DATA_BLOCK "IDB_LineC1"   // DB10
// stored: InstanceOfName LineC1.FB_LineC1, InstanceOfType FB, Namespace LineC1
"LineC1.FB_LineC1"
   // VAR
   //    "Conveyor_C1.1.1" : "Global.FB_Conveyor";
   //    "Conveyor_C1.1.2" { S7_SetPoint := 'True'} : "Global.FB_Conveyor";
   //    "Conveyor_C1.1.3" { S7_SetPoint := 'True'} : "Global.FB_Conveyor";
   //    "MABS_C1.2.1" : "Global.FB_MABS";
   //    "MABS_C1.2.2" { S7_SetPoint := 'True'} : "Global.FB_MABS";
   //    "Conveyor_C1.3.1" { S7_SetPoint := 'True'} : "Global.FB_Conveyor";
   //    "Conveyor_C1.3.2" { S7_SetPoint := 'True'} : "Global.FB_Conveyor";
   //    "Conveyor_C1.3.3" { S7_SetPoint := 'True'} : "Global.FB_Conveyor";
   //    "Conveyor_C1.3.4" { S7_SetPoint := 'True'} : "Global.FB_Conveyor";
   //    "Conveyor_C1.3.5" { S7_SetPoint := 'True'} : "Global.FB_Conveyor";
   //    "Conveyor_C1.3.6" { S7_SetPoint := 'True'} : "Global.FB_Conveyor";
   //    "Conveyor_C1.3.7" { S7_SetPoint := 'True'} : "Global.FB_Conveyor";
   //    "Conveyor_C1.3.8" { S7_SetPoint := 'True'} : "Global.FB_Conveyor";
   //    "Conveyor_C1.3.9" { S7_SetPoint := 'True'} : "Global.FB_Conveyor";
   //    "Conveyor_C1.3.10" { S7_SetPoint := 'True'} : "Global.FB_Conveyor";
   //    "Conveyor_C1.4.1" { S7_SetPoint := 'True'} : "Global.FB_Conveyor";
   //    "Conveyor_C1.4.2" { S7_SetPoint := 'True'} : "Global.FB_Conveyor";
   //    "Conveyor_C1.4.3" { S7_SetPoint := 'True'} : "Global.FB_Conveyor";
   //    "Conveyor_C1.4.4" { S7_SetPoint := 'True'} : "Global.FB_Conveyor";
   //    "Conveyor_C1.5.1" { S7_SetPoint := 'True'} : "Global.FB_Conveyor";
   //    "Conveyor_C1.6.1" { S7_SetPoint := 'True'} : "Global.FB_Conveyor";
   //    "Conveyor_C1.6.2" { S7_SetPoint := 'True'} : "Global.FB_Conveyor";
   //    "Conveyor_C1.7.1" { S7_SetPoint := 'True'} : "Global.FB_Conveyor";
   //    "Conveyor_C1.7.2" { S7_SetPoint := 'True'} : "Global.FB_Conveyor";
   //    "Conveyor_C1.7.3" { S7_SetPoint := 'True'} : "Global.FB_Conveyor";
   //    "Conveyor_C1.7.4" { S7_SetPoint := 'True'} : "Global.FB_Conveyor";
   //    "Conveyor_C1.7.5" { S7_SetPoint := 'True'} : "Global.FB_Conveyor";
   //    "Conveyor_C1.7.6" { S7_SetPoint := 'True'} : "Global.FB_Conveyor";
   //    "Conveyor_C1.7.7" { S7_SetPoint := 'True'} : "Global.FB_Conveyor";
   //    "Conveyor_C1.7.8" { S7_SetPoint := 'True'} : "Global.FB_Conveyor";
   //    "Conveyor_C1.7.9" { S7_SetPoint := 'True'} : "Global.FB_Conveyor";
   //    "Conveyor_C1.7.10" { S7_SetPoint := 'True'} : "Global.FB_Conveyor";
   //    "Conveyor_C1.8.0" { S7_SetPoint := 'True'} : "Global.FB_Conveyor";
   //    "Conveyor_C1.9.1" { S7_SetPoint := 'True'} : "Global.FB_Conveyor";
   //    "Conveyor_C1.10.1" { S7_SetPoint := 'True'} : "Global.FB_Conveyor";
   //    "Conveyor_C1.11.1" { S7_SetPoint := 'True'} : "Global.FB_Conveyor";
   //    "Conveyor_C1.11.2" { S7_SetPoint := 'True'} : "Global.FB_Conveyor";
   //    "Conveyor_C1.12.1" { S7_SetPoint := 'True'} : "Global.FB_Conveyor";
   //    "Conveyor_C1.12.2" { S7_SetPoint := 'True'} : "Global.FB_Conveyor";
   //    "Conveyor_C1.12.3" { S7_SetPoint := 'True'} : "Global.FB_Conveyor";
   //    "Transfer_C1.13.1" : "Global.FB_S300_tTransMode";
   //    "Transfer_C1.14.1" { S7_SetPoint := 'True'} : "Global.FB_S300_tTransMode";
   //    "Conveyor_C1.15.2" { S7_SetPoint := 'True'} : "Global.FB_Conveyor";
   //    "Conveyor_C1.15.3" { S7_SetPoint := 'True'} : "Global.FB_Conveyor";
   //    "Conveyor_C1.15.4" { S7_SetPoint := 'True'} : "Global.FB_Conveyor";
   //    "Conveyor_C1.16.1" { S7_SetPoint := 'True'} : "Global.FB_Conveyor";
   //    "Conveyor_C1.17.0" { S7_SetPoint := 'True'} : "Global.FB_Conveyor";
   //    "Conveyor_C1.18.1" { S7_SetPoint := 'True'} : "Global.FB_Conveyor";
   //    "Conveyor_C1.18.2" { S7_SetPoint := 'True'} : "Global.FB_Conveyor";
   //    "Conveyor_C1.18.3" { S7_SetPoint := 'True'} : "Global.FB_Conveyor";
   //    "Conveyor_C1.18.4" { S7_SetPoint := 'True'} : "Global.FB_Conveyor";
   //    "Conveyor_C1.18.5" { S7_SetPoint := 'True'} : "Global.FB_Conveyor";
   //    "Conveyor_C1.18.6" { S7_SetPoint := 'True'} : "Global.FB_Conveyor";
   //    "Conveyor_C1.18.7" { S7_SetPoint := 'True'} : "Global.FB_Conveyor";
   //    "Conveyor_C1.19.1" { S7_SetPoint := 'True'} : "Global.FB_Conveyor";
   //    "Conveyor_C1.20.2" { S7_SetPoint := 'True'} : "Global.FB_Conveyor";
   // END_VAR
BEGIN
END_DATA_BLOCK

DATA_BLOCK "IDB_LineD1"   // DB11
// stored: InstanceOfName LineD1.FB_LineD1, InstanceOfType FB, Namespace LineD1
"LineD1.FB_LineD1"
   // VAR
   //    "Conveyor_D1.1.1" : "Global.FB_Conveyor";
   //    "MABS_D1.1.1" : "Global.FB_MABS";
   //    "Transfer_D1.1.1" : "Global.FB_S300_tTransMode";
   // END_VAR
BEGIN
END_DATA_BLOCK

DATA_BLOCK "IDB_EmptyLine"   // DB9
// stored: InstanceOfName EmptyLine.FB_EmptyLine, InstanceOfType FB, Namespace EmptyLine
"EmptyLine.FB_EmptyLine"
   // VAR
   //    "J1.1.1" : "Global.FB_Conveyor";
   //    "J1.1.2" { S7_SetPoint := 'True'} : "Global.FB_Conveyor";
   //    "J1.1.3" { S7_SetPoint := 'True'} : "Global.FB_Conveyor";
   //    "J1.1.4" { S7_SetPoint := 'True'} : "Global.FB_Conveyor";
   //    "J1.1.5" { S7_SetPoint := 'True'} : "Global.FB_Conveyor";
   //    "J1.1.6" { S7_SetPoint := 'True'} : "Global.FB_Conveyor";
   //    "J1.1.7" { S7_SetPoint := 'True'} : "Global.FB_Conveyor";
   //    "J1.1.8" { S7_SetPoint := 'True'} : "Global.FB_Conveyor";
   //    "J1.1.9" { S7_SetPoint := 'True'} : "Global.FB_Conveyor";
   //    "J1.1.10" { S7_SetPoint := 'True'} : "Global.FB_Conveyor";
   //    "J1.1.11" { S7_SetPoint := 'True'} : "Global.FB_Conveyor";
   //    "J1.1.12" { S7_SetPoint := 'True'} : "Global.FB_Conveyor";
   //    "J1.1.13" { S7_SetPoint := 'True'} : "Global.FB_Conveyor";
   //    "J1.1.14" { S7_SetPoint := 'True'} : "Global.FB_Conveyor";
   //    "J1.1.15" { S7_SetPoint := 'True'} : "Global.FB_Conveyor";
   //    "J1.1.16" { S7_SetPoint := 'True'} : "Global.FB_Conveyor";
   //    "J1.2.1" { S7_SetPoint := 'True'} : "Global.FB_Conveyor";
   //    "J1.2.2" { S7_SetPoint := 'True'} : "Global.FB_Conveyor";
   //    "J1.2.3" { S7_SetPoint := 'True'} : "Global.FB_Conveyor";
   //    "J2.1.1" { S7_SetPoint := 'True'} : "Global.FB_Conveyor";
   //    "J2.1.2" { S7_SetPoint := 'True'} : "Global.FB_Conveyor";
   //    "J2.1.3" { S7_SetPoint := 'True'} : "Global.FB_Conveyor";
   //    "J2.1.4" { S7_SetPoint := 'True'} : "Global.FB_Conveyor";
   //    "J2.1.5" { S7_SetPoint := 'True'} : "Global.FB_Conveyor";
   //    "J2.1.6" { S7_SetPoint := 'True'} : "Global.FB_Conveyor";
   //    "J2.1.7" { S7_SetPoint := 'True'} : "Global.FB_Conveyor";
   //    "J2.1.8" { S7_SetPoint := 'True'} : "Global.FB_Conveyor";
   //    "J2.1.9" { S7_SetPoint := 'True'} : "Global.FB_Conveyor";
   //    "J2.1.10" { S7_SetPoint := 'True'} : "Global.FB_Conveyor";
   //    "J2.1.11" { S7_SetPoint := 'True'} : "Global.FB_Conveyor";
   //    "J2.1.12" { S7_SetPoint := 'True'} : "Global.FB_Conveyor";
   //    "J2.1.13" { S7_SetPoint := 'True'} : "Global.FB_Conveyor";
   //    "J2.1.14" { S7_SetPoint := 'True'} : "Global.FB_Conveyor";
   //    "J2.1.15" { S7_SetPoint := 'True'} : "Global.FB_Conveyor";
   //    "J2.2.1" { S7_SetPoint := 'True'} : "Global.FB_Conveyor";
   //    "J2.2.2" { S7_SetPoint := 'True'} : "Global.FB_Conveyor";
   //    "J2.3.1" { S7_SetPoint := 'True'} : "Global.FB_Conveyor";
   //    "J2.4.1" { S7_SetPoint := 'True'} : "Global.FB_Conveyor";
   //    "J1.2.4" { S7_SetPoint := 'True'} : "Global.FB_Conveyor";
   //    "J1.2.5" { S7_SetPoint := 'True'} : "Global.FB_Conveyor";
   //    "J1.3.1" { S7_SetPoint := 'True'} : "Global.FB_Conveyor";
   //    "J1.3.2" { S7_SetPoint := 'True'} : "Global.FB_Conveyor";
   //    "J1.4.1" { S7_SetPoint := 'True'} : "Global.FB_Conveyor";
   //    "J1.4.2" { S7_SetPoint := 'True'} : "Global.FB_Conveyor";
   //    "J1.4.3" { S7_SetPoint := 'True'} : "Global.FB_Conveyor";
   //    "J1.4.4" { S7_SetPoint := 'True'} : "Global.FB_Conveyor";
   //    "J1.4.5" { S7_SetPoint := 'True'} : "Global.FB_Conveyor";
   //    "J1.4.6" { S7_SetPoint := 'True'} : "Global.FB_Conveyor";
   //    "J1.4.7" { S7_SetPoint := 'True'} : "Global.FB_Conveyor";
   //    "J1.5.1" { S7_SetPoint := 'True'} : "Global.FB_Conveyor";
   //    "J1.5.2" { S7_SetPoint := 'True'} : "Global.FB_Conveyor";
   //    "J1.5.3" { S7_SetPoint := 'True'} : "Global.FB_Conveyor";
   //    "J1.5.4" { S7_SetPoint := 'True'} : "Global.FB_Conveyor";
   //    "J1.6.1" { S7_SetPoint := 'True'} : "Global.FB_MABS";
   //    "J1.6.2" { S7_SetPoint := 'True'} : "Global.FB_MABS";
   //    "J1.7.1" { S7_SetPoint := 'True'} : "Global.FB_Conveyor";
   //    "J1.7.2" { S7_SetPoint := 'True'} : "Global.FB_Conveyor";
   //    "J1.8.1" { S7_SetPoint := 'True'} : "Global.FB_Conveyor";
   //    "J1.8.2" { S7_SetPoint := 'True'} : "Global.FB_Conveyor";
   //    "J1.9.1" { S7_SetPoint := 'True'} : "Global.FB_Conveyor";
   //    "J1.10.1" { S7_SetPoint := 'True'} : "Global.FB_Conveyor";
   //    "J1.11.1" { S7_SetPoint := 'True'} : "Global.FB_Conveyor";
   //    "J1.11.2" { S7_SetPoint := 'True'} : "Global.FB_Conveyor";
   //    "J1.11.3" { S7_SetPoint := 'True'} : "Global.FB_Conveyor";
   //    "J1.11.4" { S7_SetPoint := 'True'} : "Global.FB_Conveyor";
   //    "J1.11.5" { S7_SetPoint := 'True'} : "Global.FB_Conveyor";
   //    "J1.11.6" { S7_SetPoint := 'True'} : "Global.FB_Conveyor";
   //    "J1.11.7" { S7_SetPoint := 'True'} : "Global.FB_Conveyor";
   //    "J1.11.8" { S7_SetPoint := 'True'} : "Global.FB_Conveyor";
   //    "J1.11.9" { S7_SetPoint := 'True'} : "Global.FB_Conveyor";
   //    "J1.11.10" { S7_SetPoint := 'True'} : "Global.FB_Conveyor";
   //    "J1.11.11" { S7_SetPoint := 'True'} : "Global.FB_Conveyor";
   //    "J1.11.12" { S7_SetPoint := 'True'} : "Global.FB_Conveyor";
   //    "J1.11.13" { S7_SetPoint := 'True'} : "Global.FB_Conveyor";
   //    "K1.1.1" { S7_SetPoint := 'True'} : "Global.FB_Conveyor";
   //    "K1.2.1" { S7_SetPoint := 'True'} : "Global.FB_Conveyor";
   //    "K1.3.1" { S7_SetPoint := 'True'} : "Global.FB_Conveyor";
   //    "K1.4.1" { S7_SetPoint := 'True'} : "Global.FB_Conveyor";
   //    "K1.4.2" { S7_SetPoint := 'True'} : "Global.FB_Conveyor";
   //    "K1.4.3" { S7_SetPoint := 'True'} : "Global.FB_Conveyor";
   //    "K1.4.4" { S7_SetPoint := 'True'} : "Global.FB_Conveyor";
   //    "K1.4.5" { S7_SetPoint := 'True'} : "Global.FB_Conveyor";
   //    "K1.4.6" { S7_SetPoint := 'True'} : "Global.FB_Conveyor";
   //    "K1.4.7" { S7_SetPoint := 'True'} : "Global.FB_Conveyor";
   //    "K1.4.8" { S7_SetPoint := 'True'} : "Global.FB_Conveyor";
   //    "K1.4.9" { S7_SetPoint := 'True'} : "Global.FB_Conveyor";
   //    "K1.4.10" { S7_SetPoint := 'True'} : "Global.FB_Conveyor";
   //    "K1.5.1" { S7_SetPoint := 'True'} : "Global.FB_Conveyor";
   //    "K1.5.2" { S7_SetPoint := 'True'} : "Global.FB_Conveyor";
   //    "K1.5.3" { S7_SetPoint := 'True'} : "Global.FB_Conveyor";
   //    "K1.5.4" { S7_SetPoint := 'True'} : "Global.FB_Conveyor";
   //    "K1.5.5" { S7_SetPoint := 'True'} : "Global.FB_Conveyor";
   //    "K1.5.6" { S7_SetPoint := 'True'} : "Global.FB_Conveyor";
   //    "K1.5.7" { S7_SetPoint := 'True'} : "Global.FB_Conveyor";
   //    "K1.5.8" { S7_SetPoint := 'True'} : "Global.FB_Conveyor";
   //    "K1.6.1" { S7_SetPoint := 'True'} : "Global.FB_Conveyor";
   //    "K1.6.2" { S7_SetPoint := 'True'} : "Global.FB_Conveyor";
   //    "K1.7.1" { S7_SetPoint := 'True'} : "Global.FB_Conveyor";
   //    "K1.7.2" { S7_SetPoint := 'True'} : "Global.FB_Conveyor";
   //    "K1.8.1" { S7_SetPoint := 'True'} : "Global.FB_Conveyor";
   //    "K1.8.2" { S7_SetPoint := 'True'} : "Global.FB_Conveyor";
   //    "K1.8.3" { S7_SetPoint := 'True'} : "Global.FB_Conveyor";
   //    "K1.9.1" { S7_SetPoint := 'True'} : "Global.FB_Conveyor";
   //    "K1.9.2" { S7_SetPoint := 'True'} : "Global.FB_Conveyor";
   //    "K1.9.3" { S7_SetPoint := 'True'} : "Global.FB_Conveyor";
   //    "K1.9.4" { S7_SetPoint := 'True'} : "Global.FB_Conveyor";
   //    "K1.9.5" { S7_SetPoint := 'True'} : "Global.FB_Conveyor";
   //    "K1.9.6" { S7_SetPoint := 'True'} : "Global.FB_Conveyor";
   //    "K1.9.7" { S7_SetPoint := 'True'} : "Global.FB_Conveyor";
   //    "K1.10.1" { S7_SetPoint := 'True'} : "Global.FB_Conveyor";
   // END_VAR
BEGIN
END_DATA_BLOCK

DATA_BLOCK "IDB_GlobalStatus"   // DB48
// stored: InstanceOfName Global.FB_GlobalStatus, InstanceOfType FB, Namespace Global
"Global.FB_GlobalStatus"
   // VAR
   //    Line : Struct
   //       ProductionLine : "Global.ConveyorStatus";
   //       EmptyLine { S7_SetPoint := 'True'} : "Global.ConveyorStatus";
   //       PackedLine { S7_SetPoint := 'True'} : "Global.ConveyorStatus";
   //    END_STRUCT;
   //    cmp : Struct
   //       ProductionTotes_Value0 : Array[_.gminProductionLine.._.gmaxProductionLine] of Bool;
   //       ProductionTotes_Value1 : Array[_.gminProductionLine.._.gmaxProductionLine] of Bool;
   //       EmptyLine_Value0 : Array[_.gminEmptyLine.._.gmaxEmptyLine] of Bool;
   //       EmptyLine_Value1 : Array[_.gminEmptyLine.._.gmaxEmptyLine] of Bool;
   //       PackedLine_Value0 : Array[_.gminPackedLine.._.gmaxPackedLine] of Bool;
   //       PackedLine_Value1 : Array[_.gminPackedLine.._.gmaxPackedLine] of Bool;
   //    END_STRUCT;
   //    ForVisu : Struct
   //       Line : Struct
   //          ProductionLine : Word;
   //          EmptyLine : Word;
   //          PackedLine : Word;
   //       END_STRUCT;
   //    END_STRUCT;
   // END_VAR
BEGIN
   cmp.ProductionTotes_Value1[1001..1192] := True;
   cmp.EmptyLine_Value1[2001..2109] := True;
   cmp.PackedLine_Value1[3001..3040] := True;
END_DATA_BLOCK

DATA_BLOCK "IDB_PackedLine"   // DB10
// stored: Access Published, InstanceOfName PackedLine.FB_PackedLine, InstanceOfType FB, Namespace PackedLine
"PackedLine.FB_PackedLine"
   // VAR
   //    "G1.1.1" { S7_SetPoint := 'True'} : "Global.FB_Conveyor";
   //    "G1.1.2" { S7_SetPoint := 'True'} : "Global.FB_Conveyor";
   //    "G1.1.3" { S7_SetPoint := 'True'} : "Global.FB_Conveyor";
   //    "G1.1.4" { S7_SetPoint := 'True'} : "Global.FB_Conveyor";
   //    "G1.1.5" { S7_SetPoint := 'True'} : "Global.FB_Conveyor";
   //    "G1.1.6" { S7_SetPoint := 'True'} : "Global.FB_Conveyor";
   //    "G1.1.7" { S7_SetPoint := 'True'} : "Global.FB_Conveyor";
   //    "G1.1.8" { S7_SetPoint := 'True'} : "Global.FB_Conveyor";
   //    "G1.1.9" { S7_SetPoint := 'True'} : "Global.FB_Conveyor";
   //    "G1.1.10" { S7_SetPoint := 'True'} : "Global.FB_Conveyor";
   //    "G1.1.11" { S7_SetPoint := 'True'} : "Global.FB_Conveyor";
   //    "G1.1.12" { S7_SetPoint := 'True'} : "Global.FB_Conveyor";
   //    "G1.1.13" { S7_SetPoint := 'True'} : "Global.FB_Conveyor";
   //    "G1.1.14" { S7_SetPoint := 'True'} : "Global.FB_Conveyor";
   //    "G1.1.15" { S7_SetPoint := 'True'} : "Global.FB_Conveyor";
   //    "G1.1.16" { S7_SetPoint := 'True'} : "Global.FB_Conveyor";
   //    "G1.1.17" { S7_SetPoint := 'True'} : "Global.FB_Conveyor";
   //    "G1.1.18" { S7_SetPoint := 'True'} : "Global.FB_Conveyor";
   //    "G1.1.19" { S7_SetPoint := 'True'} : "Global.FB_Conveyor";
   //    "G1.2.1" { S7_SetPoint := 'True'} : "Global.FB_Conveyor";
   //    "G1.2.2" { S7_SetPoint := 'True'} : "Global.FB_Conveyor";
   //    "G1.3.1" { S7_SetPoint := 'True'} : "Global.FB_Conveyor";
   //    "G1.4.1" { S7_SetPoint := 'True'} : "Global.FB_Conveyor";
   //    "G1.4.2" { S7_SetPoint := 'True'} : "Global.FB_Conveyor";
   //    "G1.4.3" { S7_SetPoint := 'True'} : "Global.FB_Conveyor";
   //    "G1.4.4" { S7_SetPoint := 'True'} : "Global.FB_Conveyor";
   //    "G1.4.5" { S7_SetPoint := 'True'} : "Global.FB_Conveyor";
   //    "G1.4.6" { S7_SetPoint := 'True'} : "Global.FB_Conveyor";
   //    "G1.5.1" { S7_SetPoint := 'True'} : "Global.FB_Conveyor";
   //    "G1.5.2" { S7_SetPoint := 'True'} : "Global.FB_Conveyor";
   //    "G1.5.3" { S7_SetPoint := 'True'} : "Global.FB_Conveyor";
   //    "G1.5.4" { S7_SetPoint := 'True'} : "Global.FB_Conveyor";
   //    "G1.5.5" { S7_SetPoint := 'True'} : "Global.FB_Conveyor";
   //    "G1.5.6" { S7_SetPoint := 'True'} : "Global.FB_Conveyor";
   //    "G1.6.1" { S7_SetPoint := 'True'} : "Global.FB_Conveyor";
   //    "G1.6.2" { S7_SetPoint := 'True'} : "Global.FB_Conveyor";
   //    "G1.7.1" { S7_SetPoint := 'True'} : "Global.FB_Conveyor";
   //    "G1.7.2" { S7_SetPoint := 'True'} : "Global.FB_Conveyor";
   //    "G1.7.3" { S7_SetPoint := 'True'} : "Global.FB_Conveyor";
   //    "G1.7.4" { S7_SetPoint := 'True'} : "Global.FB_Conveyor";
   // END_VAR
BEGIN
END_DATA_BLOCK

DATA_BLOCK "IDB_Merging"   // DB27
// stored: InstanceOfName ProductionLine.FB_Merging, InstanceOfType FB, Namespace ProductionLine
"ProductionLine.FB_Merging"
   // VAR
   //    "Merge_A1.7.3" : "Global.FB_Merging";
   //    "Merge_A1.9.3" : "Global.FB_Merging";
   //    "Merge_B1.6.1" { S7_SetPoint := 'True'} : "Global.FB_Merging";
   // END_VAR
BEGIN
END_DATA_BLOCK

DATA_BLOCK "IDB_ProductionLine"   // DB8
// stored: InstanceOfName ProductionLine.FB_ProductionLine, InstanceOfType FB, Namespace ProductionLine
"ProductionLine.FB_ProductionLine"
   // VAR
   //    "A1.1.1" { S7_SetPoint := 'True'} : "Global.FB_Conveyor";
   //    "A1.1.2" { S7_SetPoint := 'True'} : "Global.FB_Conveyor";
   //    "A1.1.3" { S7_SetPoint := 'True'} : "Global.FB_Conveyor";
   //    "A1.1.4" { S7_SetPoint := 'True'} : "Global.FB_Conveyor";
   //    "A1.1.5" { S7_SetPoint := 'True'} : "Global.FB_Conveyor";
   //    "A1.1.6" { S7_SetPoint := 'True'} : "Global.FB_Conveyor";
   //    "A1.1.7" { S7_SetPoint := 'True'} : "Global.FB_Conveyor";
   //    "A1.1.8" { S7_SetPoint := 'True'} : "Global.FB_Conveyor";
   //    "A1.1.9" { S7_SetPoint := 'True'} : "Global.FB_Conveyor";
   //    "A1.1.10" { S7_SetPoint := 'True'} : "Global.FB_Conveyor";
   //    "A1.1.11" { S7_SetPoint := 'True'} : "Global.FB_Conveyor";
   //    "A1.1.12" { S7_SetPoint := 'True'} : "Global.FB_Conveyor";
   //    "A1.1.13" { S7_SetPoint := 'True'} : "Global.FB_Conveyor";
   //    "A1.1.14" { S7_SetPoint := 'True'} : "Global.FB_Conveyor";
   //    "A1.2.1" { S7_SetPoint := 'True'} : "Global.FB_Conveyor";
   //    "A1.3.1" { S7_SetPoint := 'True'} : "Global.FB_Conveyor";
   //    "A1.4.1" { S7_SetPoint := 'True'} : "Global.FB_Conveyor";
   //    "A1.5.1" { S7_SetPoint := 'True'} : "Global.FB_Conveyor";
   //    "A1.5.2" { S7_SetPoint := 'True'} : "Global.FB_Conveyor";
   //    "A1.5.3" { S7_SetPoint := 'True'} : "Global.FB_Conveyor";
   //    "A1.7.1" { S7_SetPoint := 'True'} : "Global.FB_Conveyor";
   //    "A1.7.2" { S7_SetPoint := 'True'} : "Global.FB_Conveyor";
   //    "A1.7.3" { S7_SetPoint := 'True'} : "Global.FB_Conveyor";
   //    "A1.7.4" { S7_SetPoint := 'True'} : "Global.FB_Conveyor";
   //    "A1.7.5" { S7_SetPoint := 'True'} : "Global.FB_Conveyor";
   //    "A1.7.6" { S7_SetPoint := 'True'} : "Global.FB_Conveyor";
   //    "A1.8.1" { S7_SetPoint := 'True'} : "Global.FB_Conveyor";
   //    "A1.10.1" { S7_SetPoint := 'True'} : "Global.FB_Conveyor";
   //    "A1.10.2" { S7_SetPoint := 'True'} : "Global.FB_Conveyor";
   //    "A1.10.3" { S7_SetPoint := 'True'} : "Global.FB_Conveyor";
   //    "A1.10.4" { S7_SetPoint := 'True'} : "Global.FB_Conveyor";
   //    "A1.10.5" { S7_SetPoint := 'True'} : "Global.FB_Conveyor";
   //    "A1.10.6" { S7_SetPoint := 'True'} : "Global.FB_Conveyor";
   //    "A1.10.7" { S7_SetPoint := 'True'} : "Global.FB_Conveyor";
   //    "A1.10.8" { S7_SetPoint := 'True'} : "Global.FB_Conveyor";
   //    "A1.10.9" { S7_SetPoint := 'True'} : "Global.FB_Conveyor";
   //    "A1.10.10" { S7_SetPoint := 'True'} : "Global.FB_Conveyor";
   //    "A1.10.11" { S7_SetPoint := 'True'} : "Global.FB_Conveyor";
   //    "A1.10.12" { S7_SetPoint := 'True'} : "Global.FB_Conveyor";
   //    "A1.10.13" { S7_SetPoint := 'True'} : "Global.FB_Conveyor";
   //    "A1.11.1" { S7_SetPoint := 'True'} : "Global.FB_Conveyor";
   //    "A1.11.2" { S7_SetPoint := 'True'} : "Global.FB_Conveyor";
   //    "A1.12.1" { S7_SetPoint := 'True'} : "Global.FB_Conveyor";
   //    "A1.12.2" { S7_SetPoint := 'True'} : "Global.FB_Conveyor";
   //    "A1.14.1" { S7_SetPoint := 'True'} : "Global.FB_Conveyor";
   //    "A1.14.2" { S7_SetPoint := 'True'} : "Global.FB_Conveyor";
   //    "A1.14.3" { S7_SetPoint := 'True'} : "Global.FB_Conveyor";
   //    "A1.14.4" { S7_SetPoint := 'True'} : "Global.FB_Conveyor";
   //    "A1.14.5" { S7_SetPoint := 'True'} : "Global.FB_Conveyor";
   //    "A1.14.6" { S7_SetPoint := 'True'} : "Global.FB_Conveyor";
   //    "A1.14.7" { S7_SetPoint := 'True'} : "Global.FB_Conveyor";
   //    "A1.14.8" { S7_SetPoint := 'True'} : "Global.FB_Conveyor";
   //    "A1.14.9" { S7_SetPoint := 'True'} : "Global.FB_Conveyor";
   //    "A1.14.10" { S7_SetPoint := 'True'} : "Global.FB_Conveyor";
   //    "A1.14.11" { S7_SetPoint := 'True'} : "Global.FB_Conveyor";
   //    "A1.14.12" { S7_SetPoint := 'True'} : "Global.FB_Conveyor";
   //    "A1.14.13" { S7_SetPoint := 'True'} : "Global.FB_Conveyor";
   //    "A1.14.14" { S7_SetPoint := 'True'} : "Global.FB_Conveyor";
   //    "A1.14.15" { S7_SetPoint := 'True'} : "Global.FB_Conveyor";
   //    "A1.14.16" { S7_SetPoint := 'True'} : "Global.FB_Conveyor";
   //    "A1.14.17" { S7_SetPoint := 'True'} : "Global.FB_Conveyor";
   //    "A1.14.18" { S7_SetPoint := 'True'} : "Global.FB_Conveyor";
   //    "A1.14.19" { S7_SetPoint := 'True'} : "Global.FB_Conveyor";
   //    "A1.14.20" { S7_SetPoint := 'True'} : "Global.FB_Conveyor";
   //    "A1.14.21" { S7_SetPoint := 'True'} : "Global.FB_Conveyor";
   //    "A1.14.22" { S7_SetPoint := 'True'} : "Global.FB_Conveyor";
   //    "A1.14.23" { S7_SetPoint := 'True'} : "Global.FB_Conveyor";
   //    "A1.14.24" { S7_SetPoint := 'True'} : "Global.FB_Conveyor";
   //    "A1.14.25" { S7_SetPoint := 'True'} : "Global.FB_Conveyor";
   //    "A1.14.26" { S7_SetPoint := 'True'} : "Global.FB_Conveyor";
   //    "A2.2.1" { S7_SetPoint := 'True'} : "Global.FB_Conveyor";
   //    "A2.2.2" { S7_SetPoint := 'True'} : "Global.FB_Conveyor";
   //    "A2.2.3" { S7_SetPoint := 'True'} : "Global.FB_Conveyor";
   //    "A2.2.4" { S7_SetPoint := 'True'} : "Global.FB_Conveyor";
   //    "A2.2.5" { S7_SetPoint := 'True'} : "Global.FB_Conveyor";
   //    "A2.2.6" { S7_SetPoint := 'True'} : "Global.FB_Conveyor";
   //    "A2.2.7" { S7_SetPoint := 'True'} : "Global.FB_Conveyor";
   //    "A2.2.8" { S7_SetPoint := 'True'} : "Global.FB_Conveyor";
   //    "A2.2.9" { S7_SetPoint := 'True'} : "Global.FB_Conveyor";
   //    "A2.2.10" { S7_SetPoint := 'True'} : "Global.FB_Conveyor";
   //    "A2.2.11" { S7_SetPoint := 'True'} : "Global.FB_Conveyor";
   //    "A2.2.12" { S7_SetPoint := 'True'} : "Global.FB_Conveyor";
   //    "A2.2.13" { S7_SetPoint := 'True'} : "Global.FB_Conveyor";
   //    "A2.2.14" { S7_SetPoint := 'True'} : "Global.FB_Conveyor";
   //    "A2.2.15" { S7_SetPoint := 'True'} : "Global.FB_Conveyor";
   //    "A2.2.16" { S7_SetPoint := 'True'} : "Global.FB_Conveyor";
   //    "A2.2.17" { S7_SetPoint := 'True'} : "Global.FB_Conveyor";
   //    "A2.2.18" { S7_SetPoint := 'True'} : "Global.FB_Conveyor";
   //    "A2.2.19" { S7_SetPoint := 'True'} : "Global.FB_Conveyor";
   //    "A2.2.20" { S7_SetPoint := 'True'} : "Global.FB_Conveyor";
   //    "A2.2.21" { S7_SetPoint := 'True'} : "Global.FB_Conveyor";
   //    "A2.2.22" { S7_SetPoint := 'True'} : "Global.FB_Conveyor";
   //    "A2.2.23" { S7_SetPoint := 'True'} : "Global.FB_Conveyor";
   //    "A2.2.24" { S7_SetPoint := 'True'} : "Global.FB_Conveyor";
   //    "A2.2.25" { S7_SetPoint := 'True'} : "Global.FB_Conveyor";
   //    "A2.2.26" { S7_SetPoint := 'True'} : "Global.FB_Conveyor";
   //    "B1.1.1" { S7_SetPoint := 'True'} : "Global.FB_Conveyor";
   //    "B1.2.1" { S7_SetPoint := 'True'} : "Global.FB_Conveyor";
   //    "B1.3.1" { S7_SetPoint := 'True'} : "Global.FB_Conveyor";
   //    "B1.3.2" { S7_SetPoint := 'True'} : "Global.FB_Conveyor";
   //    "B1.3.3" { S7_SetPoint := 'True'} : "Global.FB_Conveyor";
   //    "B1.4.1" { S7_SetPoint := 'True'} : "Global.FB_Conveyor";
   //    "B1.4.2" { S7_SetPoint := 'True'} : "Global.FB_Conveyor";
   //    "B1.5.1" { S7_SetPoint := 'True'} : "Global.FB_Conveyor";
   //    "B1.7.1" { S7_SetPoint := 'True'} : "Global.FB_Conveyor";
   //    "B1.7.2" { S7_SetPoint := 'True'} : "Global.FB_Conveyor";
   //    "B1.7.3" { S7_SetPoint := 'True'} : "Global.FB_Conveyor";
   //    "B1.8.1" { S7_SetPoint := 'True'} : "Global.FB_Conveyor";
   //    "B1.8.2" { S7_SetPoint := 'True'} : "Global.FB_Conveyor";
   //    "B1.8.3" { S7_SetPoint := 'True'} : "Global.FB_Conveyor";
   //    "B1.9.1" { S7_SetPoint := 'True'} : "Global.FB_Conveyor";
   //    "B1.9.2" { S7_SetPoint := 'True'} : "Global.FB_Conveyor";
   //    "B1.11.1" { S7_SetPoint := 'True'} : "Global.FB_Conveyor";
   //    "B1.11.2" { S7_SetPoint := 'True'} : "Global.FB_Conveyor";
   //    "B1.11.3" { S7_SetPoint := 'True'} : "Global.FB_Conveyor";
   //    "B1.11.4" { S7_SetPoint := 'True'} : "Global.FB_Conveyor";
   //    "B1.12.1" { S7_SetPoint := 'True'} : "Global.FB_Conveyor";
   //    "B1.12.2" { S7_SetPoint := 'True'} : "Global.FB_Conveyor";
   //    "B1.15.1" { S7_SetPoint := 'True'} : "Global.FB_Conveyor";
   //    "B1.15.2" { S7_SetPoint := 'True'} : "Global.FB_Conveyor";
   //    "B1.16.1" { S7_SetPoint := 'True'} : "Global.FB_Conveyor";
   //    "B1.16.2" { S7_SetPoint := 'True'} : "Global.FB_Conveyor";
   //    "B1.16.3" { S7_SetPoint := 'True'} : "Global.FB_Conveyor";
   //    "B1.16.4" { S7_SetPoint := 'True'} : "Global.FB_Conveyor";
   //    "B1.16.5" { S7_SetPoint := 'True'} : "Global.FB_Conveyor";
   //    "B1.16.6" { S7_SetPoint := 'True'} : "Global.FB_Conveyor";
   //    "B1.16.7" { S7_SetPoint := 'True'} : "Global.FB_Conveyor";
   //    "B1.16.8" { S7_SetPoint := 'True'} : "Global.FB_Conveyor";
   //    "B1.17.1" { S7_SetPoint := 'True'} : "Global.FB_Conveyor";
   //    "B1.17.2" { S7_SetPoint := 'True'} : "Global.FB_Conveyor";
   //    "B1.17.3" { S7_SetPoint := 'True'} : "Global.FB_Conveyor";
   //    "B1.17.4" { S7_SetPoint := 'True'} : "Global.FB_Conveyor";
   //    "B1.19.1" { S7_SetPoint := 'True'} : "Global.FB_Conveyor";
   //    "B1.20.1" { S7_SetPoint := 'True'} : "Global.FB_Conveyor";
   //    "B1.20.2" { S7_SetPoint := 'True'} : "Global.FB_Conveyor";
   //    "B1.21.1" { S7_SetPoint := 'True'} : "Global.FB_Conveyor";
   //    "B1.21.2" { S7_SetPoint := 'True'} : "Global.FB_Conveyor";
   //    "B1.21.3" { S7_SetPoint := 'True'} : "Global.FB_Conveyor";
   //    "B1.22.1" { S7_SetPoint := 'True'} : "Global.FB_Conveyor";
   //    "B1.23.1" { S7_SetPoint := 'True'} : "Global.FB_Conveyor";
   //    "C1.2.2" { S7_SetPoint := 'True'} : "Global.FB_Conveyor";
   //    "C1.2.1" { S7_SetPoint := 'True'} : "Global.FB_Conveyor";
   //    "C1.4.1" { S7_SetPoint := 'True'} : "Global.FB_Conveyor";
   //    "C1.4.2" { S7_SetPoint := 'True'} : "Global.FB_Conveyor";
   //    "D1.1.1" { S7_SetPoint := 'True'} : "Global.FB_Conveyor";
   //    "D1.2.1" { S7_SetPoint := 'True'} : "Global.FB_Conveyor";
   //    "D1.3.1" { S7_SetPoint := 'True'} : "Global.FB_Conveyor";
   //    "D1.4.1" { S7_SetPoint := 'True'} : "Global.FB_Conveyor";
   //    "D1.5.1" { S7_SetPoint := 'True'} : "Global.FB_Conveyor";
   //    "D1.6.1" { S7_SetPoint := 'True'} : "Global.FB_Conveyor";
   //    "D1.7.1" { S7_SetPoint := 'True'} : "Global.FB_Conveyor";
   //    "D1.7.2" { S7_SetPoint := 'True'} : "Global.FB_Conveyor";
   //    "D1.7.3" { S7_SetPoint := 'True'} : "Global.FB_Conveyor";
   //    "D1.7.4" { S7_SetPoint := 'True'} : "Global.FB_Conveyor";
   //    "D1.7.5" { S7_SetPoint := 'True'} : "Global.FB_Conveyor";
   //    "D1.7.6" { S7_SetPoint := 'True'} : "Global.FB_Conveyor";
   //    "D1.7.7" { S7_SetPoint := 'True'} : "Global.FB_Conveyor";
   //    "D1.7.8" { S7_SetPoint := 'True'} : "Global.FB_Conveyor";
   //    "D1.7.9" { S7_SetPoint := 'True'} : "Global.FB_Conveyor";
   //    "D1.7.10" { S7_SetPoint := 'True'} : "Global.FB_Conveyor";
   //    "D1.8.1" { S7_SetPoint := 'True'} : "Global.FB_Conveyor";
   //    "D1.8.2" { S7_SetPoint := 'True'} : "Global.FB_Conveyor";
   //    "D1.8.3" { S7_SetPoint := 'True'} : "Global.FB_Conveyor";
   //    "D1.11.1" { S7_SetPoint := 'True'} : "Global.FB_Conveyor";
   //    "D1.11.2" { S7_SetPoint := 'True'} : "Global.FB_Conveyor";
   //    "D1.11.3" { S7_SetPoint := 'True'} : "Global.FB_Conveyor";
   //    "D1.12.1" { S7_SetPoint := 'True'} : "Global.FB_Conveyor";
   //    "D1.12.2" { S7_SetPoint := 'True'} : "Global.FB_Conveyor";
   //    "D1.12.3" { S7_SetPoint := 'True'} : "Global.FB_Conveyor";
   //    "E1.1.1" { S7_SetPoint := 'True'} : "Global.FB_Conveyor";
   //    "E1.1.2" { S7_SetPoint := 'True'} : "Global.FB_Conveyor";
   //    "E1.1.3" { S7_SetPoint := 'True'} : "Global.FB_Conveyor";
   //    "E1.1.4" { S7_SetPoint := 'True'} : "Global.FB_Conveyor";
   //    "E1.2.1" { S7_SetPoint := 'True'} : "Global.FB_Conveyor";
   //    "E1.3.1" { S7_SetPoint := 'True'} : "Global.FB_Conveyor";
   //    "E1.4.1" { S7_SetPoint := 'True'} : "Global.FB_Conveyor";
   //    "E1.5.1" { S7_SetPoint := 'True'} : "Global.FB_Conveyor";
   //    "E1.6.1" { S7_SetPoint := 'True'} : "Global.FB_Conveyor";
   //    "A1.9.1" { S7_SetPoint := 'True'} : "Global.FB_MABS";
   //    "A1.9.2" { S7_SetPoint := 'True'} : "Global.FB_MABS";
   //    "A1.6.1" { S7_SetPoint := 'True'} : "Global.FB_MABS";
   //    "A1.6.2" { S7_SetPoint := 'True'} : "Global.FB_MABS";
   //    "A1.13.1" { S7_SetPoint := 'True'} : "Global.FB_S300_tTransMode";
   //    "A2.1.1" { S7_SetPoint := 'True'} : "Global.FB_S300_tTransMode";
   //    "B1.6.1" { S7_SetPoint := 'True'} : "Global.FB_S300_FullControl";
   //    "B1.10.1" { S7_SetPoint := 'True'} : "Global.FB_S300_tTransMode";
   //    "B1.13.1" { S7_SetPoint := 'True'} : "Global.FB_S300_tTransMode";
   //    "B1.14.1" { S7_SetPoint := 'True'} : "Global.FB_S300_tTransMode";
   //    "B1.18.1" { S7_SetPoint := 'True'} : "Global.FB_S300_tTransMode";
   //    "C1.3.1" { S7_SetPoint := 'True'} : "Global.FB_S300_tTransMode";
   //    "D1.9.2" { S7_SetPoint := 'True'} : "Global.FB_S300_tTransMode";
   //    "D1.10.1" { S7_SetPoint := 'True'} : "Global.FB_S300_tTransMode";
   // END_VAR
BEGIN
END_DATA_BLOCK

DATA_BLOCK "IDB_VisuAlarm"   // DB49
// stored: Access Published, InstanceOfName Global.FB_VisuAlarm, InstanceOfType FB, Namespace Global
"Global.FB_VisuAlarm"
   // VAR
   //    noAlarmState : Bool;
   //    CommunicationFault : Struct
   //       PLC : Word;
   //       "BW-ASi" : Word;
   //       Cognex : Word;
   //       Mabs : Word;
   //    END_STRUCT;
   //    "BW-ASi" : Struct
   //       "BW_ASi143 -MCC100 -210KE3 -ConfigErr_Circuit1_Slave(0-15)A_1" : Word;
   //       "BW_ASi143 -MCC100 -210KE3 -ConfigErr_Circuit1_Slave(16-31)A" : Word;
   //       "BW_ASi143 -MCC100 -210KE3 -ConfigErr_Circuit1_Slave(0-15)B_1" : Word;
   //       "BW_ASi143 -MCC100 -210KE3 -ConfigErr_Circuit1_Slave(16-31)B" : Word;
   //       "BW_ASi143 -MCC100 -210KE3 -PeriErr_Circuit1_Slave(0-15)A_1" : Word;
   //       "BW_ASi143 -MCC100 -210KE3 -PeriErr_Circuit1_Slave(16-31)A" : Word;
   //       "BW_ASi143 -MCC100 -210KE3 -PeriErr_Circuit1_Slave(0-15)B_1" : Word;
   //       "BW_ASi143 -MCC100 -210KE3 -PeriErr_Circuit1_Slave(16-31)B" : Word;
   //       "BW_ASi143 -MCC100 -210KE3 -ConfigErr_Circuit2_Slave(0-15)A" : Word;
   //       "BW_ASi143 -MCC100 -210KE3 -ConfigErr_Circuit2_Slave(16-31)A" : Word;
   //       "BW_ASi143 -MCC100 -210KE3 -ConfigErr_Circuit2_Slave(0-15)B" : Word;
   //       "BW_ASi143 -MCC100 -210KE3 -ConfigErr_Circuit2_Slave(16-31)B" : Word;
   //       "BW_ASi143 -MCC100 -210KE3 -PeriErr_Circuit2_Slave(0-15)A" : Word;
   //       "BW_ASi143 -MCC100 -210KE3 -PeriErr_Circuit2_Slave(16-31)A" : Word;
   //       "BW_ASi143 -MCC100 -210KE3 -PeriErr_Circuit2_Slave(0-15)B" : Word;
   //       "BW_ASi143 -MCC100 -210KE3 -PeriErr_Circuit2_Slave(16-31)B" : Word;
   //       "BW_ASi200 -MCC300 -210KE3 -ConfigErr_Circuit1_Slave(0-15)A" : Word;
   //       "BW_ASi200 -MCC300 -210KE3 -ConfigErr_Circuit1_Slave(16-31)A" : Word;
   //       "BW_ASi200 -MCC300 -210KE3 -ConfigErr_Circuit1_Slave(0-15)B" : Word;
   //       "BW_ASi200 -MCC300 -210KE3 -ConfigErr_Circuit1_Slave(16-31)B" : Word;
   //       "BW_ASi200 -MCC300 -210KE3 -PeriErr_Circuit1_Slave(0-15)A" : Word;
   //       "BW_ASi200 -MCC300 -210KE3 -PeriErr_Circuit1_Slave(16-31)A" : Word;
   //       "BW_ASi200 -MCC300 -210KE3 -PeriErr_Circuit1_Slave(0-15)B" : Word;
   //       "BW_ASi200 -MCC300 -210KE3 -PeriErr_Circuit1_Slave(16-31)B" : Word;
   //       "BW_ASi200 -MCC300 -210KE3 -ConfigErr_Circuit2_Slave(0-15)A" : Word;
   //       "BW_ASi200 -MCC300 -210KE3 -ConfigErr_Circuit2_Slave(16-31)A" : Word;
   //       "BW_ASi200 -MCC300 -210KE3 -ConfigErr_Circuit2_Slave(0-15)B" : Word;
   //       "BW_ASi200 -MCC300 -210KE3 -ConfigErr_Circuit2_Slave(16-31)B" : Word;
   //       "BW_ASi200 -MCC300 -210KE3 -PeriErr_Circuit2_Slave(0-15)A" : Word;
   //       "BW_ASi200 -MCC300 -210KE3 -PeriErr_Circuit2_Slave(16-31)A" : Word;
   //       "BW_ASi200 -MCC300 -210KE3 -PeriErr_Circuit2_Slave(0-15)B" : Word;
   //       "BW_ASi200 -MCC300 -210KE3 -PeriErr_Circuit2_Slave(16-31)B" : Word;
   //    END_STRUCT;
   //    "word" : Struct
   //       Line : Struct
   //          ProductionLine : Struct
   //             Conveyor : Array[_.gminProductionLine.._.gmaxProductionLine] of Word;
   //          END_STRUCT;
   //          EmptyLine : Struct
   //             Conveyor : Array[_.gminEmptyLine.._.gmaxEmptyLine] of Word;
   //          END_STRUCT;
   //          PackedLine : Struct
   //             Conveyor : Array[_.gminPackedLine.._.gmaxPackedLine] of Word;
   //          END_STRUCT;
   //       END_STRUCT;
   //    END_STRUCT;
   // END_VAR
BEGIN
END_DATA_BLOCK

DATA_BLOCK "IDB_DataMan262"   // DB40
// stored: InstanceOfName Global.DataMan262, InstanceOfType FB, Namespace Global
"Global.DataMan262"
   // VAR_INPUT
   //    TriggerSignal : Bool;
   //    ContinuousGetResults : Bool;
   //    "Dataman-Results Available" : Bool;
   //    "Dataman-TriggerReady" : Bool;
   //    "Dataman-TriggerAck" : Bool;
   //    "Dataman-Train Focus Ack" : Bool;
   //    "Dataman-Train Match String Ack" : Bool;
   //    "Dataman-Execute DMCC Ack" : Bool;
   //    "Dataman-Set Match String Ack" : Bool;
   //    "Dataman-ResultID" : Int;
   //    "Dataman-Result Code" : Int;
   //    "Dataman-Result Length" : Int;
   //    "Result Data" : "Global.BarCode";
   // END_VAR
   // VAR_OUTPUT
   //    "Dataman-UserData Length" : Word;
   //    "Dataman-UserData Option" : Word;
   //    "User Data" : "Global.BarCode";
   // END_VAR
   // VAR_IN_OUT
   //    "Dataman-TriggerEnable" : Bool;
   //    "Dataman-Trigger" : Bool;
   //    "Dataman-ResultsAck" : Bool;
   //    "Dataman-Train Focus" : Bool;
   //    "Dataman-Train Match String" : Bool;
   //    "Dataman-Execute DMCC" : Bool;
   //    "Dataman-Set Match String" : Bool;
   // END_VAR
   // VAR
   //    "Result Pending" : Bool;
   //    "Latest Results" : Struct
   //       ID : Int;
   //       Flags : Int;
   //       Length : Int;
   //       Value : Array[0..63] of Byte;
   //    END_STRUCT;
   //    "Train Focus" : Bool;
   //    "Train MatchString" : Bool;
   //    "Execute DMCC" : Bool;
   //    "Set Match String" : Bool;
   //    "String" : String[64];
   //    "Match String" : Array[0..63] of Byte;
   //    "Char" : Array[0..63] of Byte;
   //    Ret_val_1 { ExternalAccessible := 'False'; ExternalVisible := 'False'; ExternalWritable := 'False'} : Byte;
   //    R_TRIG_SimpleRead { S7_SetPoint := 'True'} : R_TRIG;
   //    R_TRIG_TrainFocus { S7_SetPoint := 'True'} : R_TRIG;
   //    "R_TRIG_Train MatchString" { S7_SetPoint := 'True'} : R_TRIG;
   //    R_TRIG_ExcuteDMCC { S7_SetPoint := 'True'} : R_TRIG;
   //    R_TRIG_SetMatchString { S7_SetPoint := 'True'} : R_TRIG;
   //    HoldTrigger { S7_SetPoint := 'True'} : Bool;
   //    HoldTrainFocus : Bool;
   //    HoldTrainMatchString : Bool;
   //    HoldDMCCExcute : Bool;
   //    HoldSetMatchString : Bool;
   // END_VAR
BEGIN
END_DATA_BLOCK

DATA_BLOCK "IDB_FB_Merging"   // DB39
// stored: InstanceOfName LineC1.FB_Merging, InstanceOfType FB, Namespace LineC1
"LineC1.FB_Merging"
   // VAR
   //    Merge : "Global.FB_Merging";
   // END_VAR
BEGIN
END_DATA_BLOCK

DATA_BLOCK "IDB_ManualControl"   // DB50
// stored: InstanceOfName Global.FB_ManualControl, InstanceOfType FB, Namespace Global
"Global.FB_ManualControl"
   // VAR RETAIN
   //    "Counter" { S7_SetPoint := 'True'} : CTU_INT;
   // END_VAR
BEGIN
END_DATA_BLOCK

DATA_BLOCK "IDB_Flow_Test"   // DB46
// stored: InstanceOfName ProductionLine.Flow_Test, InstanceOfType FB, Namespace ProductionLine
"ProductionLine.Flow_Test"
   // VAR
   //    Start { S7_SetPoint := 'True'} : Bool;
   //    StartTest { S7_SetPoint := 'True'} : "ProductionLine.Test_Logic";
   //    GoToRightDP1 { S7_SetPoint := 'True'} : "ProductionLine.Test_Logic";
   //    ContinueStraightDP1 { S7_SetPoint := 'True'} : "ProductionLine.Test_Logic";
   //    ContinueStraightDP2 { S7_SetPoint := 'True'} : "ProductionLine.Test_Logic";
   //    GotorightDP2Thentoright { S7_SetPoint := 'True'} : "ProductionLine.Test_Logic";
   //    GotorightDP2ThentoLeft { S7_SetPoint := 'True'} : "ProductionLine.Test_Logic";
   //    ContinueStraightDP3 { S7_SetPoint := 'True'} : "ProductionLine.Test_Logic";
   //    ContinueStraightDP4 { S7_SetPoint := 'True'} : "ProductionLine.Test_Logic";
   //    GotoRightDP4 { S7_SetPoint := 'True'} : "ProductionLine.Test_Logic";
   //    "A1.13.1_Straight" { S7_SetPoint := 'True'} : "ProductionLine.Test_Logic";
   //    "A1.13.1_left" { S7_SetPoint := 'True'} : "ProductionLine.Test_Logic";
   //    R_TRIG_Instance { S7_SetPoint := 'True'} : R_TRIG;
   // END_VAR
BEGIN
END_DATA_BLOCK

DATA_BLOCK "IDB_FB_ToggleDir"   // DB47
// stored: InstanceOfName ProductionLine.FB_ToggleDir, InstanceOfType FB, Namespace ProductionLine
"ProductionLine.FB_ToggleDir"
   // VAR
   //    "A1.12.1" { S7_SetPoint := 'True'} : "Global.ToggelDir";
   //    CurrentExpedtionDirection : Struct
   //       Straight : Bool;
   //       Left : Bool;
   //       None : Bool;
   //    END_STRUCT;
   //    CurrentStraightTableselection : Struct
   //       Table1 : Bool;
   //       Table2 : Bool;
   //       Table3 : Bool;
   //       Table4 : Bool;
   //       Table5 : Bool;
   //       None : Bool;
   //    END_STRUCT;
   //    CurrentLeftTableselection : Struct
   //       Table1 : Bool;
   //       Table2 : Bool;
   //       Table3 : Bool;
   //       Table4 : Bool;
   //       Table5 : Bool;
   //       None : Bool;
   //    END_STRUCT;
   // END_VAR
BEGIN
END_DATA_BLOCK

DATA_BLOCK "IDB_BarcodeReader"   // DB29
// stored: InstanceOfName ProductionLine.BarcodeReader, InstanceOfType FB, Namespace ProductionLine
"ProductionLine.BarcodeReader"
   // VAR
   //    DP1 : "Global.DataMan262";
   //    DP2 : "Global.DataMan262";
   //    DP3 : "Global.DataMan262";
   //    DP4 : "Global.DataMan262";
   // END_VAR
BEGIN
END_DATA_BLOCK

DATA_BLOCK "IDB_FB_Technology"   // DB38
// stored: InstanceOfName ProductionLine.FB_Technology, InstanceOfType FB, Namespace ProductionLine
"ProductionLine.FB_Technology"
   // VAR
   //    IP11 : String;
   //    IP12 : String;
   //    IP21 : String;
   //    IP22 : String;
   //    IP23 : String;
   //    IP31 : String;
   //    IP32 : String;
   //    IP41 : String;
   //    IP42 : String;
   //    ComDownStream : Struct
   //       DP1 : Bool;
   //       DP2 : Bool;
   //       DP3 : Bool;
   //       DP4 : Bool;
   //    END_STRUCT;
   //    ComTimmerDP1 { S7_SetPoint := 'True'} : TON_TIME;
   //    ComTimmerDP2 { S7_SetPoint := 'True'} : TON_TIME;
   //    ComTimmerDP3 { S7_SetPoint := 'True'} : TON_TIME;
   //    ComTimmerDP4 { S7_SetPoint := 'True'} : TON_TIME;
   // END_VAR
BEGIN
END_DATA_BLOCK

DATA_BLOCK "IDB_OPC_Communication"   // DB42
// stored: InstanceOfName ProductionLine.FB_OPC_Communication, InstanceOfType FB, Namespace ProductionLine
"ProductionLine.FB_OPC_Communication"
   // VAR
   //    Communication_DP1 : "ProductionLine.FB_OPC_DestRequest";
   //    Communication_DP2 : "ProductionLine.FB_OPC_DestRequest";
   //    Communication_DP3 : "ProductionLine.FB_OPC_DestRequest";
   //    Communication_DP4 : "ProductionLine.FB_OPC_DestRequest";
   //    Communication_IP1 : "ProductionLine.FB_OPC_DestInfo";
   //    Communication_IP2 : "ProductionLine.FB_OPC_DestInfo";
   //    Communication_IP3 : "ProductionLine.FB_OPC_DestInfo";
   //    Communication_IP4 : "ProductionLine.FB_OPC_DestInfo";
   //    Communication_IP5 : "ProductionLine.FB_OPC_DestInfo";
   //    Communication_IP6 : "ProductionLine.FB_OPC_DestInfo";
   //    Communication_IP7 : "ProductionLine.FB_OPC_DestInfo";
   //    Communication_IP8 : "ProductionLine.FB_OPC_DestInfo";
   //    Communication_IP9 : "ProductionLine.FB_OPC_DestInfo";
   //    Communication_SYS_OP : "ProductionLine.FB_OPC_SysStatus";
   //    Communication_SYS_OP_Source { S7_SetPoint := 'True'} : "ProductionLine.OPC_SystemStatus";
   //    Communication_SYS_OP_Ack { S7_SetPoint := 'True'} : "ProductionLine.OPC_SystStatus_Ack";
   //    timPeriodicSend { S7_SetPoint := 'True'} : IEC_TIMER;
   //    timWatchdog { S7_SetPoint := 'True'} : IEC_TIMER;
   //    Communication_fault : Bool;
   // END_VAR
BEGIN
END_DATA_BLOCK

DATA_BLOCK "IDB_Segments_Status"   // DB45
// stored: InstanceOfName ProductionLine.FB_Segments, InstanceOfType FB, Namespace ProductionLine
"ProductionLine.FB_Segments"
   // VAR
   //    ConveyorID : Int;
   //    "Counter" : Int;
   //    FlowRackLoop1 : Array[_."B1.1.1".._."B1.23.1"] of Bool;
   //    FlowRackLoop2 : Array[_."B1.6.1".._."B1.18.1"] of Bool;
   //    Fragileloop1 : Array[_."D1.1.1".._."E1.6.1"] of Bool;
   //    Fragileloop2 : Array[_."D1.9.1".._."D1.10.1"] of Bool;
   //    cmp : Struct
   //       FlowRackLoop1 : Array[_."B1.1.1".._."B1.23.1"] of Bool;
   //       FlowRackLoop2 : Array[_."B1.6.1".._."B1.18.1"] of Bool;
   //       Fragileloop1 : Array[_."D1.1.1".._."E1.6.1"] of Bool;
   //       Fragileloop2 : Array[_."D1.9.1".._."D1.10.1"] of Bool;
   //    END_STRUCT;
   //    FlowRackLoopReadyToRun : Bool;
   //    FlowRackWorkPlaceLeftReadyToRun : Bool;
   //    FlowRackWorkPlaceRightReadyToRun : Bool;
   //    FragileloopReadyToRun : Bool;
   // END_VAR
BEGIN
END_DATA_BLOCK

DATA_BLOCK "IDB_ToteTracking"   // DB11
// stored: InstanceOfName ProductionLine.FB_ToteTracking, InstanceOfType FB, Namespace ProductionLine
"ProductionLine.FB_ToteTracking"
   // VAR
   //    ZoneBpJam_Occ : TON_TIME;
   //    ZoneBpJam_NotOcc { S7_SetPoint := 'True'} : TON_TIME;
   //    DivertToManual { S7_SetPoint := 'True'} : Bool;
   //    HoldDivertToManual : Bool;
   //    RT_Exit_1_ : Array[1..1] of R_TRIG;
   //    RT_Exit_2_ : Array[1..6] of R_TRIG;
   //    NoReadTote { S7_SetPoint := 'True'} : String;
   //    NoData : Array[1..6] of Bool;
   // END_VAR
BEGIN
END_DATA_BLOCK
